Fanuc KAREL source: port_UOUT.kl

PROGRAM TP
%NOLOCKGROUP
VAR
 x: BOOLEAN
BEGIN
 x = UOUT[3]
END TP
